ABB RAPID module: final.prg

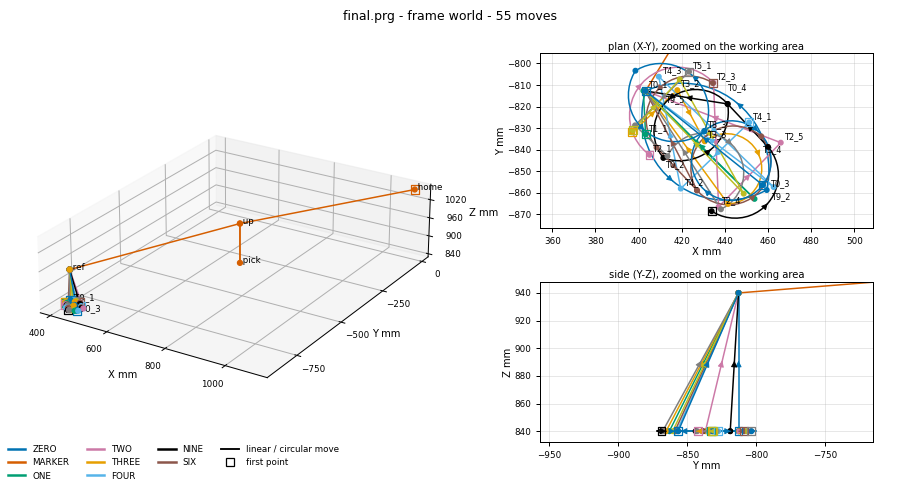
[picture p0: tool path of final.prg in frame world, 55 of 55 moves have a stored position in this frame; points joined in program order, loops and branches not executed]
MODULE Module1
    PERS tooldata Efector:=[TRUE,[[0,0.033033672,184.3],[1,0,0,0]],[1.5,[0,0,90],[1,0,0,0],0.01,0.01,0.01]];
    PERS wobjdata Workobject_1:=[FALSE,TRUE,"",[[276.123735704,-827.667234537,798.663444233],[0.923877305,0.000104396,-0.002651392,-0.382679612]],[[0,0,0],[1,0,0,0]]];
    CONST robtarget T0_1:=[[79.546208479,100.497907125,40.730455604],[0.002409616,-0.000002677,-0.99999648,0.001111092],[-1,-1,0,0],[9E+09,9E+09,9E+09,9E+09,9E+09,9E+09]];
    CONST robtarget T0_2:=[[111.035842809,79.777621062,40.624742502],[0.002409616,-0.000002677,-0.99999648,0.001111092],[-1,-1,0,0],[9E+09,9E+09,9E+09,9E+09,9E+09,9E+09]];
    CONST robtarget T0_3:=[[151.732370203,107.749116179,40.366456021],[0.002409616,-0.000002677,-0.99999648,0.001111092],[-1,-1,0,0],[9E+09,9E+09,9E+09,9E+09,9E+09,9E+09]];
    CONST robtarget T0_4:=[[106.187899089,125.180560875,40.547211878],[0.002409616,-0.000002677,-0.99999648,0.001111092],[-1,-1,0,0],[9E+09,9E+09,9E+09,9E+09,9E+09,9E+09]];
    CONST robtarget home:=[[0.834488103,1170.696929347,259.084700159],[0.459642479,-0.331462463,0.801426912,0.191249396],[-1,0,-1,0],[9E+09,9E+09,9E+09,9E+09,9E+09,9E+09]];
    CONST robtarget up:=[[-51.633208179,640.397645531,178.164826806],[0.705400436,-0.000783768,0.708808148,-0.000787554],[-1,-2,1,0],[9E+09,9E+09,9E+09,9E+09,9E+09,9E+09]];
    CONST robtarget pick:=[[-52.259706896,640.108764023,48.166657408],[0.705400436,-0.000783768,0.708808148,-0.000787554],[-1,-2,1,0],[9E+09,9E+09,9E+09,9E+09,9E+09,9E+09]];
    CONST robtarget ref:=[[80.028130577,100.720123453,140.72904745],[0.002409616,-0.000002677,-0.99999648,0.001111092],[-1,0,-1,0],[9E+09,9E+09,9E+09,9E+09,9E+09,9E+09]];
    CONST robtarget T1_1:=[[93.778043214,86.267789909,40.693490346],[0.002409616,-0.000002677,-0.99999648,0.001111093],[-1,0,-1,0],[9E+09,9E+09,9E+09,9E+09,9E+09,9E+09]];
    CONST robtarget T1_2:=[[78.731217939,99.845917516,40.735832074],[0.002409616,-0.000002677,-0.99999648,0.001111093],[-1,0,-1,0],[9E+09,9E+09,9E+09,9E+09,9E+09,9E+09]];
    CONST robtarget T1_3:=[[150.636382929,100.842145042,40.387086501],[0.002409616,-0.000002677,-0.99999648,0.001111093],[-1,0,-1,0],[9E+09,9E+09,9E+09,9E+09,9E+09,9E+09]];
    CONST robtarget T2_1:=[[101.755950553,80.841717855,40.667100297],[0.002409616,-0.000002677,-0.99999648,0.001111093],[-1,0,-1,0],[9E+09,9E+09,9E+09,9E+09,9E+09,9E+09]];
    CONST robtarget T2_2:=[[76.08624864,99.311947147,40.74976553],[0.002409616,-0.000002677,-0.99999648,0.001111093],[-1,0,-1,0],[9E+09,9E+09,9E+09,9E+09,9E+09,9E+09]];
    CONST robtarget T2_3:=[[99.104981321,125.470636052,40.580701845],[0.002409616,-0.000002677,-0.99999648,0.001111093],[-1,0,-1,0],[9E+09,9E+09,9E+09,9E+09,9E+09,9E+09]];
    CONST robtarget T2_4:=[[141.480489244,86.448278602,40.463197375],[0.002409616,-0.000002677,-0.99999648,0.001111093],[-1,0,-1,0],[9E+09,9E+09,9E+09,9E+09,9E+09,9E+09]];
    CONST robtarget T2_5:=[[140.80349709,127.872183573,40.374407927],[0.002409616,-0.000002677,-0.99999648,0.001111093],[-1,0,-1,0],[9E+09,9E+09,9E+09,9E+09,9E+09,9E+09]];
    CONST robtarget T3_1:=[[88.710215411,82.591773594,40.726082499],[0.002409616,-0.000002677,-0.99999648,0.001111093],[-1,0,-1,0],[9E+09,9E+09,9E+09,9E+09,9E+09,9E+09]];
    CONST robtarget T3_2:=[[89.688090682,111.187772163,40.657823899],[0.002409616,-0.000002677,-0.99999648,0.001111093],[-1,0,-1,0],[9E+09,9E+09,9E+09,9E+09,9E+09,9E+09]];
    CONST robtarget T3_3:=[[115.419791871,103.366515913,40.55119576],[0.002409616,-0.000002677,-0.99999648,0.001111093],[-1,0,-1,0],[9E+09,9E+09,9E+09,9E+09,9E+09,9E+09]];
    CONST robtarget T3_4:=[[138.022529389,116.554241299,40.41296091],[0.002409616,-0.000002677,-0.99999648,0.001111093],[-1,0,-1,0],[9E+09,9E+09,9E+09,9E+09,9E+09,9E+09]];
    CONST robtarget T3_5:=[[143.635464218,90.505245507,40.443796548],[0.002409616,-0.000002677,-0.99999648,0.001111093],[-1,0,-1,0],[9E+09,9E+09,9E+09,9E+09,9E+09,9E+09]];
    CONST robtarget T4_1:=[[123.83069419,124.165374487,40.464442032],[0.002409616,-0.000002677,-0.99999648,0.001111093],[-1,0,-1,0],[9E+09,9E+09,9E+09,9E+09,9E+09,9E+09]];
    CONST robtarget T4_2:=[[123.075702975,80.033491537,40.566150282],[0.002409616,-0.000002677,-0.99999648,0.001111093],[-1,0,-1,0],[9E+09,9E+09,9E+09,9E+09,9E+09,9E+09]];
    CONST robtarget T4_3:=[[79.18787321,109.525888713,40.712120516],[0.002409616,-0.000002677,-0.99999648,0.001111093],[-1,0,-1,0],[9E+09,9E+09,9E+09,9E+09,9E+09,9E+09]];
    CONST robtarget T4_4:=[[153.035355052,110.99609425,40.352961057],[0.002409616,-0.000002677,-0.99999648,0.001111093],[-1,0,-1,0],[9E+09,9E+09,9E+09,9E+09,9E+09,9E+09]];
    CONST robtarget T9_1:=[[140.611499337,82.764297004,40.475571821],[0.002409616,-0.000002677,-0.99999648,0.001111093],[-1,0,-1,0],[9E+09,9E+09,9E+09,9E+09,9E+09,9E+09]];
    CONST robtarget T9_2:=[[156.448315421,103.968075054,40.352130656],[0.002409616,-0.000002677,-0.99999648,0.001111093],[-1,0,-1,0],[9E+09,9E+09,9E+09,9E+09,9E+09,9E+09]];
    CONST robtarget T9_3:=[[138.016529456,122.326227112,40.400163337],[0.002409616,-0.000002677,-0.99999648,0.001111093],[-1,0,-1,0],[9E+09,9E+09,9E+09,9E+09,9E+09,9E+09]];
    CONST robtarget T9_4:=[[110.69684671,123.155517631,40.529981942],[0.002409616,-0.000002677,-0.99999648,0.001111093],[-1,0,-1,0],[9E+09,9E+09,9E+09,9E+09,9E+09,9E+09]];
    CONST robtarget T9_5:=[[90.029086726,101.021793612,40.678771345],[0.002409616,-0.000002677,-0.99999648,0.001111093],[-1,0,-1,0],[9E+09,9E+09,9E+09,9E+09,9E+09,9E+09]];
    CONST robtarget T9_6:=[[107.315885986,84.371649598,40.632461157],[0.002409616,-0.000002677,-0.99999648,0.001111093],[-1,0,-1,0],[9E+09,9E+09,9E+09,9E+09,9E+09,9E+09]];
    CONST robtarget T9_7:=[[119.971739012,101.45747188,40.533500882],[0.002409616,-0.000002677,-0.99999648,0.001111093],[-1,0,-1,0],[9E+09,9E+09,9E+09,9E+09,9E+09,9E+09]];
    CONST robtarget T6_1:=[[99.037119424,125.16526603,40.581707484],[0.002409616,0.000002677,-0.99999648,0.001111093],[-1,-1,-1,0],[9E+09,9E+09,9E+09,9E+09,9E+09,9E+09]];
    CONST robtarget T6_2:=[[83.20030334,103.96148798,40.705148627],[0.002409616,0.000002677,-0.99999648,0.001111093],[-1,-1,-1,0],[9E+09,9E+09,9E+09,9E+09,9E+09,9E+09]];
    CONST robtarget T6_3:=[[101.632089305,85.603335922,40.657115952],[0.002409616,0.000002677,-0.99999648,0.001111093],[-1,-1,-1,0],[9E+09,9E+09,9E+09,9E+09,9E+09,9E+09]];
    CONST robtarget T6_4:=[[128.951772051,84.774045403,40.527297366],[0.002409616,0.000002677,-0.99999648,0.001111093],[-1,-1,-1,0],[9E+09,9E+09,9E+09,9E+09,9E+09,9E+09]];
    CONST robtarget T6_5:=[[149.619532035,106.907769422,40.378507987],[0.002409616,0.000002677,-0.99999648,0.001111093],[-1,-1,-1,0],[9E+09,9E+09,9E+09,9E+09,9E+09,9E+09]];
    CONST robtarget T6_6:=[[132.332732775,123.557913436,40.424818171],[0.002409616,0.000002677,-0.99999648,0.001111093],[-1,-1,-1,0],[9E+09,9E+09,9E+09,9E+09,9E+09,9E+09]];
    CONST robtarget T6_7:=[[114.189479584,106.472149918,40.550223668],[0.002409616,0.000002677,-0.99999648,0.001111093],[-1,-1,-1,0],[9E+09,9E+09,9E+09,9E+09,9E+09,9E+09]];
    CONST robtarget T5_1:=[[87.47494015,121.068036328,40.646533482],[0.002409616,-0.000002677,-0.99999648,0.001111092],[-1,0,-1,0],[9E+09,9E+09,9E+09,9E+09,9E+09,9E+09]];
    CONST robtarget T5_2:=[[87.358941509,85.796124659,40.725473626],[0.002409616,-0.000002677,-0.99999648,0.001111092],[-1,0,-1,0],[9E+09,9E+09,9E+09,9E+09,9E+09,9E+09]];
    CONST robtarget T5_3:=[[108.084700828,86.30490145,40.62445961],[0.002409616,-0.000002677,-0.99999648,0.001111092],[-1,0,-1,0],[9E+09,9E+09,9E+09,9E+09,9E+09,9E+09]];
    CONST robtarget T5_4:=[[126.476487242,111.192166678,40.480519899],[0.002409616,-0.000002677,-0.99999648,0.001111092],[-1,0,-1,0],[9E+09,9E+09,9E+09,9E+09,9E+09,9E+09]];
    CONST robtarget T5_5:=[[143.027295052,86.419526967,40.455806449],[0.002409616,-0.000002677,-0.99999648,0.001111092],[-1,0,-1,0],[9E+09,9E+09,9E+09,9E+09,9E+09,9E+09]];
    CONST robtarget T7_1:=[[88.254137879,83.451889647,40.726368808],[0.002409616,-0.000002677,-0.99999648,0.001111092],[-1,0,-1,0],[9E+09,9E+09,9E+09,9E+09,9E+09,9E+09]];
    CONST robtarget T7_2:=[[86.933153208,115.512476931,40.661490103],[0.002409616,-0.000002677,-0.99999648,0.001111092],[-1,0,-1,0],[9E+09,9E+09,9E+09,9E+09,9E+09,9E+09]];
    CONST robtarget T7_3:=[[145.380474485,98.997889493,40.416514244],[0.002409616,-0.000002677,-0.99999648,0.001111092],[-1,0,-1,0],[9E+09,9E+09,9E+09,9E+09,9E+09,9E+09]];
    CONST robtarget T8_1:=[[148.856287686,108.091037322,40.379556329],[0.002409616,-0.000002677,-0.99999648,0.001111092],[-1,0,-1,0],[9E+09,9E+09,9E+09,9E+09,9E+09,9E+09]];
    CONST robtarget T8_2:=[[127.493535772,87.570316763,40.528110688],[0.002409616,-0.000002677,-0.99999648,0.001111092],[-1,0,-1,0],[9E+09,9E+09,9E+09,9E+09,9E+09,9E+09]];
    CONST robtarget T8_3:=[[111.951716246,106.624436154,40.560669208],[0.002409616,-0.000002677,-0.99999648,0.001111092],[-1,0,-1,0],[9E+09,9E+09,9E+09,9E+09,9E+09,9E+09]];
    CONST robtarget T8_4:=[[88.719986023,120.847649824,40.641022855],[0.002409616,-0.000002677,-0.99999648,0.001111092],[-1,0,-1,0],[9E+09,9E+09,9E+09,9E+09,9E+09,9E+09]];
    CONST robtarget T8_5:=[[69.565208467,103.81389701,40.771187619],[0.002409616,-0.000002677,-0.99999648,0.001111092],[-1,0,-1,0],[9E+09,9E+09,9E+09,9E+09,9E+09,9E+09]];
    CONST robtarget T8_6:=[[90.170969186,87.149717488,40.708913585],[0.002409616,-0.000002677,-0.99999648,0.001111092],[-1,0,-1,0],[9E+09,9E+09,9E+09,9E+09,9E+09,9E+09]];
    CONST robtarget T8_7:=[[130.168504694,124.215197637,40.433787102],[0.002409616,-0.000002677,-0.99999648,0.001111092],[-1,0,-1,0],[9E+09,9E+09,9E+09,9E+09,9E+09,9E+09]];

    PROC main()
        MARKER;
        ZERO;
    ENDPROC


    PROC ZERO()
        MoveL T0_1,v200,fine,Efector\WObj:=Workobject_1;
        MoveC T0_2,T0_3,v200,fine,Efector\WObj:=Workobject_1;
        MoveC T0_4,T0_1,v200,fine,Efector\WObj:=Workobject_1;
        MoveL ref,v200,fine,Efector\WObj:=Workobject_1;
    ENDPROC
    PROC MARKER()
        Set DO10_9;
        MoveL home,v200,fine,Efector\WObj:=Workobject_1;
        MoveL up,v200,fine,Efector\WObj:=Workobject_1;
        MoveL pick,v200,fine,Efector\WObj:=Workobject_1;
        Reset DO10_9;
        WaitTime 2;
        MoveL up,v200,fine,Efector\WObj:=Workobject_1;
        WaitTime 2;
        MoveL ref,v200,fine,Efector\WObj:=Workobject_1;
    ENDPROC
    PROC ONE()
        MoveL T1_1,v200,fine,Efector\WObj:=Workobject_1;
        MoveL T1_2,v200,fine,Efector\WObj:=Workobject_1;
        MoveL T1_3,v200,fine,Efector\WObj:=Workobject_1;
        MoveL ref,v200,fine,Efector\WObj:=Workobject_1;
    ENDPROC
    PROC TWO()
        MoveL T2_1,v200,fine,Efector\WObj:=Workobject_1;
        MoveC T2_2,T2_3,v200,fine,Efector\WObj:=Workobject_1;
        MoveL T2_4,v200,fine,Efector\WObj:=Workobject_1;
        MoveL T2_5,v200,fine,Efector\WObj:=Workobject_1;
        MoveL ref,v200,fine,Efector\WObj:=Workobject_1;
    ENDPROC
    PROC THREE()
        MoveL T3_1,v200,fine,Efector\WObj:=Workobject_1;
        MoveL T3_2,v200,fine,Efector\WObj:=Workobject_1;
        MoveL T3_3,v200,fine,Efector\WObj:=Workobject_1;
        MoveC T3_4,T3_5,v200,fine,Efector\WObj:=Workobject_1;
        MoveL ref,v200,fine,Efector\WObj:=Workobject_1;
    ENDPROC
    PROC FOUR()
        MoveL T4_1,v200,fine,Efector\WObj:=Workobject_1;
        MoveL T4_2,v200,fine,Efector\WObj:=Workobject_1;
        MoveL T4_3,v200,fine,Efector\WObj:=Workobject_1;
        MoveL T4_4,v200,fine,Efector\WObj:=Workobject_1;
        MoveL ref,v200,fine,Efector\WObj:=Workobject_1;
    ENDPROC
    PROC NINE()
        MoveL T9_1,v200,fine,Efector\WObj:=Workobject_1;
        MoveC T9_2,T9_3,v200,fine,Efector\WObj:=Workobject_1;
        MoveL T9_4,v200,fine,Efector\WObj:=Workobject_1;
        MoveC T9_5,T9_6,v200,fine,Efector\WObj:=Workobject_1;
        MoveC T9_7,T9_4,v200,fine,Efector\WObj:=Workobject_1;
        MoveL ref,v200,fine,Efector\WObj:=Workobject_1;
    ENDPROC
    PROC SIX()
        MoveL T6_1,v200,fine,Efector\WObj:=Workobject_1;
        MoveC T6_2,T6_3,v200,fine,Efector\WObj:=Workobject_1;
        MoveL T6_4,v200,fine,Efector\WObj:=Workobject_1;
        MoveC T6_5,T6_6,v200,fine,Efector\WObj:=Workobject_1;
        MoveC T6_7,T6_4,v200,fine,Efector\WObj:=Workobject_1;
        MoveL ref,v200,fine,Efector\WObj:=Workobject_1;
    ENDPROC
    PROC FIVE()
        MoveL T5_1,v200,fine,Efector\WObj:=Workobject_1;
        MoveL T5_2,v200,fine,Efector\WObj:=Workobject_1;
        MoveL T5_3,v200,fine,Efector\WObj:=Workobject_1;
        MoveC T5_4,T5_5,v200,fine,Efector\WObj:=Workobject_1;
        MoveL ref,v200,fine,Efector\WObj:=Workobject_1;
    ENDPROC
    PROC SEVEN()
        MoveL T7_1,v200,fine,Efector\WObj:=Workobject_1;
        MoveL T7_2,v200,fine,Efector\WObj:=Workobject_1;
        MoveL T7_3,v200,fine,Efector\WObj:=Workobject_1;
        MoveL ref,v200,fine,Efector\WObj:=Workobject_1;
    ENDPROC
    PROC EIGHT()
        MoveL T8_1,v200,fine,Efector\WObj:=Workobject_1;
        MoveC T8_2,T8_3,v200,fine,Efector\WObj:=Workobject_1;
        MoveC T8_4,T8_5,v200,fine,Efector\WObj:=Workobject_1;
        MoveC T8_6,T8_3,v200,fine,Efector\WObj:=Workobject_1;
        MoveC T8_7,T8_1,v200,fine,Efector\WObj:=Workobject_1;
        MoveL ref,v200,fine,Efector\WObj:=Workobject_1;
    ENDPROC
ENDMODULE
